# EPICS substitutions: labjack/labjackApp/Db/labjack_T7_bi.substitutions
file "labjack_t7_bi.template"
{
 pattern
{ P	, R			, In			, Bit	, DESC			, ZNAM		, ONAM		, ZSV		, OSV		, SCAN		}
{ Depo	, "{}"
}
